# EPICS substitutions: ek9000App/Db/EL3072.substitutions
file EL3072.template
{       pattern
        {
                TERMINAL,

        }
        {
        }
}
